// TIA Portal V16 export
// export: Created 2021-04-13T11:10:15.6852195Z, ExportSetting WithDefaults, DisplayName Totally Integrated Automation Portal, DisplayVersion V16, DisplayName TIA Portal Version Control Interface, DisplayVersion V16, DisplayName TIA Portal Openness, DisplayVersion V16, DisplayName STEP 7 Professional, DisplayVersion V16, DisplayName STEP 7 Safety, DisplayVersion V16, DisplayName WinCC Unified SCADA Engineering System, DisplayVersion V16
DATA_BLOCK "hmi"   // DB200
{ S7_Optimized_Access := 'FALSE' }
VERSION : 0.1
// stored: AutoNumber false, DBAccessibleFromOPCUA true, IsOnlyStoredInLoadMemory false, IsWriteProtectedInAS false
   VAR
      alarmTest : "alarmsPlant";
      autoMode : Bool;   // автоматический режим
      isEnableAutoMode : Bool;
      calibrWeightMode : "calibrationModule";   // калибровка и тарирование весов
      dataStantion : "dataStantion";
      manRunAllVibroLot : Bool;
      manStopAllVibroLot : Bool;
      NewReadyWeightOnLine : Array[0..12] of Bool;
      outConvAndPack : Array[0..2] of "outConv";
      permitOn1Bunk : Array[0..12] of Bool;
      permitOn2Bunk : Array[0..12] of Bool;
      plavnik : "plavnik";
      readySystem : Int;
      recipeVar : "recipeVar";   // переменные рецепта
      rotary : "rotary";   // анимация вращения конвейеров
      sourceConv : "sourceConv";
      timeWorkConvAuto : Int;
      weightLine : Array[0..12] of "LineWeight";
      currentSetRecipes : String := '$00$00';
      numPage : Int;
      commonAlarm : Bool;   // Сигнал если хотябы одна авария есть
      report : Struct
         perfomance : Int;   // производительность
         sumPreWeight : Real;   // суммарная переработка веса
         commonTimeWork : Real;   // время работы установки
      END_STRUCT;
      addedVibro : "addedVibro";
   END_VAR
BEGIN
   // alarmTest.bit[0] : Управляющие цепи деактивированны
   // alarmTest.bit[1] : весовой модуль не в сети 1
   // alarmTest.bit[2] : весовой модуль не в сети 2
   // alarmTest.bit[3] : весовой модуль не в сети 3
   // alarmTest.bit[4] : весовой модуль не в сети 4
   // alarmTest.bit[5] : весовой модуль не в сети 5
   // alarmTest.bit[6] : весовой модуль не в сети 6
   // alarmTest.bit[7] : весовой модуль не в сети 7
   // alarmTest.bit[8] : весовой модуль не в сети 8
   // alarmTest.bit[9] : весовой модуль не в сети 9
   // alarmTest.bit[10] : весовой модуль не в сети 10
   // alarmTest.bit[11] : весовой модуль не в сети 11
   // alarmTest.bit[12] : весовой модуль не в сети 12
   // alarmTest.bit[13] : обрыв датчик весового модуля 1 -значение выше 7000
   // alarmTest.bit[14] : обрыв датчик весового модуля 2
   // alarmTest.bit[15] : обрыв датчик весового модуля 3
   // alarmTest.bit[16] : обрыв датчик весового модуля 4
   // alarmTest.bit[17] : обрыв датчик весового модуля 5
   // alarmTest.bit[18] : обрыв датчик весового модуля 6
   // alarmTest.bit[19] : обрыв датчик весового модуля 7
   // alarmTest.bit[20] : обрыв датчик весового модуля 8
   // alarmTest.bit[21] : обрыв датчик весового модуля 9
   // alarmTest.bit[22] : обрыв датчик весового модуля 10
   // alarmTest.bit[23] : обрыв датчик весового модуля 11
   // alarmTest.bit[24] : обрыв датчик весового модуля 12
   // alarmTest.bit[25] : Напряжение сети не в норме
   // alarmTest.bit[26] : Тепловое реле Конв1
   // alarmTest.bit[27] : тепловое реле Конв2
   // alarmTest.bit[58] : Нажат аварийный пост
   // alarmTest.bit[59] : Авария бункер 1
   // alarmTest.bit[60] : Авария бункер 2
   // alarmTest.bit[61] : Авария бункер 3
   // alarmTest.bit[62] : Авария бункер 4
   // alarmTest.bit[63] : Авария бункер 5
   // alarmTest.bit[64] : Авария бункер 6
   // alarmTest.bit[65] : Авария бункер 7
   // alarmTest.bit[66] : Авария бункер 8
   // alarmTest.bit[67] : Авария бункер 9
   // alarmTest.bit[68] : Авария бункер 10
   // alarmTest.bit[69] : Авария бункер 11
   // alarmTest.bit[70] : Авария бункер 12
   // alarmTest.bit[80] : сброс таймера моточасов
   // alarmTest.bit[81] : датчик просвета
   // alarmTest.bit[83] : Нет возможности сформировать порцию
   // calibrWeightMode.calib : калибровка весов
   // calibrWeightMode.tara : тарирование весов
END_DATA_BLOCK
